{attribute addProperty BoxType "EK1100-0000-0018"}
{attribute addProperty Id "Beckhoff_EL3xxxEK1122Beckhoff_EL3xxxEK1122_9FE29313162A_0001_EL3602_0000_0016EL3602_174E163625832.25A_0002_EL3602_0000_0017EL3602_174E163625832.25A_0003_EL3602_0000_0018EL3602_174E163625832.25A_0004_EL3602_0000_0019EL3602_174E163625832.25A_0005_EL3602_0002_0016EL3602_338E185817822.25A_0006_EL3602_0002_0017EL3602_338E185817822.25A_0007_EL3602_0002_0018EL3602_338E185817822.25A_0008_EL3602_0010_0016EL3602_174E163625832.25A_0009_EL3602_0010_0017EL3602_174E163625832.25A_0010_EL3602_0010_0018EL3602_174E163625832.25A_0011_EL3602_0010_0019EL3602_174E163625832.25A_0012_EL3602_0020_0018EL3602_5DBFB1A027634.5A_0013_EL3611_1030_0016EL3611_AB57A9CF13016.25A_0014_EL3611_1030_0017EL3611_AB57A9CF13016.25A_0015_EL3612_0000_0016EL3612_174E163625832.25A_0016_EL3612_0000_0017EL3612_174E163625832.25A_0017_EL3612_0000_0018EL3612_174E163625832.25A_0018_EL3612_0000_0019EL3612_174E163625832.25A_0019_EL3612_0020_0018EL3612_174E163625832.25A_0020_EL3612_0020_0019EL3612_174E163625832.25A_0021_EL3621_0020_0016EL3621_336DEF4513016.25A_0022_EL3621_0020_0017EL3621_336DEF4513016.25A_0023_EL3632_0000_0016EL3632_D178097B57872.25A_0024_EL3632_0000_0017EL3632_D178097B57872.25A_0025_EL3632_0000_0018EL3632_D178097B57872.25A_0026_EL3632_0000_0019EL3632_D178097B57872.25A_0027_EL3632_0000_0020EL3632_D178097B57872.25A_0028_EL3632_0000_0021EL3632_D178097B57872.25A_0029_EL3632_0000_0022EL3632_A724E07457872.25A_0030_EL3632_0000_0023EL3632_A724E07457872.25A_0031_EL3681_0000_0017EL3681_0CFA3F6116220.25A_0032_EL3681_0000_0018EL3681_BC5DB35D16220.25A_0033_EL3681_0000_0019EL3681_BC5DB35D16220.25A_0034_EL3681_0000_0020EL3681_C596F5D116220.25A_0035_EL3681_0000_0021EL3681_AB553B5016220.25A_0036_EL3692_0000_0017EL3692_0443616427434.25A_0037_EL3692_0000_0018EL3692_0443616427434.25A_0038_EL3692_0000_0019EL3692_0443616427434.25A_0039_EL3692_0000_0020EL3692_4E8506B127434.25A_0040_EL3692_0000_0021EL3692_4E8506B127434.25"}
{attribute addProperty CRC "1753762497"}
{attribute addProperty SizeInBites "11762"}
{attribute addProperty SizeInBytes "1470.25"}
TYPE Beckhoff_EL3xxx_68884AC1 EXTENDS EK1100_179A0949 :
STRUCT
	{attribute addProperty Name "Beckhoff_EL3xxxEK1122"}
	Beckhoff_EL3xxxEK1122 : Beckhoff_EL3xxxEK1122_9FE29313;
	{attribute addProperty Name "A_0001_EL3602_0000_0016"}
	A_0001_EL3602_0000_0016 : EL3602_174E1636;
	{attribute addProperty Name "A_0002_EL3602_0000_0017"}
	A_0002_EL3602_0000_0017 : EL3602_174E1636;
	{attribute addProperty Name "A_0003_EL3602_0000_0018"}
	A_0003_EL3602_0000_0018 : EL3602_174E1636;
	{attribute addProperty Name "A_0004_EL3602_0000_0019"}
	A_0004_EL3602_0000_0019 : EL3602_174E1636;
	{attribute addProperty Name "A_0005_EL3602_0002_0016"}
	A_0005_EL3602_0002_0016 : EL3602_338E1858;
	{attribute addProperty Name "A_0006_EL3602_0002_0017"}
	A_0006_EL3602_0002_0017 : EL3602_338E1858;
	{attribute addProperty Name "A_0007_EL3602_0002_0018"}
	A_0007_EL3602_0002_0018 : EL3602_338E1858;
	{attribute addProperty Name "A_0008_EL3602_0010_0016"}
	A_0008_EL3602_0010_0016 : EL3602_174E1636;
	{attribute addProperty Name "A_0009_EL3602_0010_0017"}
	A_0009_EL3602_0010_0017 : EL3602_174E1636;
	{attribute addProperty Name "A_0010_EL3602_0010_0018"}
	A_0010_EL3602_0010_0018 : EL3602_174E1636;
	{attribute addProperty Name "A_0011_EL3602_0010_0019"}
	A_0011_EL3602_0010_0019 : EL3602_174E1636;
	{attribute addProperty Name "A_0012_EL3602_0020_0018"}
	A_0012_EL3602_0020_0018 : EL3602_5DBFB1A0;
	{attribute addProperty Name "A_0013_EL3611_1030_0016"}
	A_0013_EL3611_1030_0016 : EL3611_AB57A9CF;
	{attribute addProperty Name "A_0014_EL3611_1030_0017"}
	A_0014_EL3611_1030_0017 : EL3611_AB57A9CF;
	{attribute addProperty Name "A_0015_EL3612_0000_0016"}
	A_0015_EL3612_0000_0016 : EL3612_174E1636;
	{attribute addProperty Name "A_0016_EL3612_0000_0017"}
	A_0016_EL3612_0000_0017 : EL3612_174E1636;
	{attribute addProperty Name "A_0017_EL3612_0000_0018"}
	A_0017_EL3612_0000_0018 : EL3612_174E1636;
	{attribute addProperty Name "A_0018_EL3612_0000_0019"}
	A_0018_EL3612_0000_0019 : EL3612_174E1636;
	{attribute addProperty Name "A_0019_EL3612_0020_0018"}
	A_0019_EL3612_0020_0018 : EL3612_174E1636;
	{attribute addProperty Name "A_0020_EL3612_0020_0019"}
	A_0020_EL3612_0020_0019 : EL3612_174E1636;
	{attribute addProperty Name "A_0021_EL3621_0020_0016"}
	A_0021_EL3621_0020_0016 : EL3621_336DEF45;
	{attribute addProperty Name "A_0022_EL3621_0020_0017"}
	A_0022_EL3621_0020_0017 : EL3621_336DEF45;
	{attribute addProperty Name "A_0023_EL3632_0000_0016"}
	A_0023_EL3632_0000_0016 : EL3632_D178097B;
	{attribute addProperty Name "A_0024_EL3632_0000_0017"}
	A_0024_EL3632_0000_0017 : EL3632_D178097B;
	{attribute addProperty Name "A_0025_EL3632_0000_0018"}
	A_0025_EL3632_0000_0018 : EL3632_D178097B;
	{attribute addProperty Name "A_0026_EL3632_0000_0019"}
	A_0026_EL3632_0000_0019 : EL3632_D178097B;
	{attribute addProperty Name "A_0027_EL3632_0000_0020"}
	A_0027_EL3632_0000_0020 : EL3632_D178097B;
	{attribute addProperty Name "A_0028_EL3632_0000_0021"}
	A_0028_EL3632_0000_0021 : EL3632_D178097B;
	{attribute addProperty Name "A_0029_EL3632_0000_0022"}
	A_0029_EL3632_0000_0022 : EL3632_A724E074;
	{attribute addProperty Name "A_0030_EL3632_0000_0023"}
	A_0030_EL3632_0000_0023 : EL3632_A724E074;
	{attribute addProperty Name "A_0031_EL3681_0000_0017"}
	A_0031_EL3681_0000_0017 : EL3681_0CFA3F61;
	{attribute addProperty Name "A_0032_EL3681_0000_0018"}
	A_0032_EL3681_0000_0018 : EL3681_BC5DB35D;
	{attribute addProperty Name "A_0033_EL3681_0000_0019"}
	A_0033_EL3681_0000_0019 : EL3681_BC5DB35D;
	{attribute addProperty Name "A_0034_EL3681_0000_0020"}
	A_0034_EL3681_0000_0020 : EL3681_C596F5D1;
	{attribute addProperty Name "A_0035_EL3681_0000_0021"}
	A_0035_EL3681_0000_0021 : EL3681_AB553B50;
	{attribute addProperty Name "A_0036_EL3692_0000_0017"}
	A_0036_EL3692_0000_0017 : EL3692_04436164;
	{attribute addProperty Name "A_0037_EL3692_0000_0018"}
	A_0037_EL3692_0000_0018 : EL3692_04436164;
	{attribute addProperty Name "A_0038_EL3692_0000_0019"}
	A_0038_EL3692_0000_0019 : EL3692_04436164;
	{attribute addProperty Name "A_0039_EL3692_0000_0020"}
	A_0039_EL3692_0000_0020 : EL3692_4E8506B1;
	{attribute addProperty Name "A_0040_EL3692_0000_0021"}
	A_0040_EL3692_0000_0021 : EL3692_4E8506B1;
END_STRUCT
END_TYPE

(* stored: Version 1.2.0.0, ProductVersion 3.1.4024.9
   DUT Beckhoff_EL3xxx_68884AC1: Id {62883086-6317-4ac2-a91b-c1e011f4c4c6} *)
